// Mitsubishi GX Works2 project: plc_group_3   PLC: FX3G
// 20.11 דורין

// global labels: Global1
VAR_GLOBAL
  START_DAY AT Y010 : BOOL;
  START_WASHING AT X002 : BOOL;
  TS_200 AT TS200 : BOOL;
  Y_5 AT Y005 : BOOL;
  TC_200 AT TC200 : BOOL;
END_VAR
VAR_GLOBAL CONSTANT
  TIMER_1 : INT := 300;
  ORANGE_VALUE : REAL;
END_VAR
VAR_GLOBAL
  ORANGE AT D1270 : REAL;
  ORANGE_STOCK AT D1110 : REAL;  (* ORANGE STOCK *)
  POMELO AT D1280 : REAL;  (* POMELO *)
  POMELO_STOCK AT D1119 : REAL;  (* POMELO *)
  CLAMENTINE AT D1275 : REAL;  (* CLEMENTINE STOCK *)
  CLAMENTINE_wasing AT D1112 : REAL;  (* CLEMENTINE STOCK *)
  POMELO_washing AT D1122 : REAL;  (* POMELO *)
  ORANGE_washing AT D1155 : REAL;
  check_orange_amount AT X020 : BOOL;
  washig_empty AT D1230 : REAL;  (* POMELO *)
  if_more_than_100 AT D1165 : INT;
END_VAR
VAR_GLOBAL CONSTANT
  ORANGES_100 : INT := 100;
END_VAR
VAR_GLOBAL
  OUTPUT_oranges AT D1130 : INT;
  cc_0 AT CC0 : BOOL;
END_VAR
VAR_GLOBAL CONSTANT
  k_2 : WORD := 2;
END_VAR
VAR_GLOBAL
  m_0 AT M0 : BOOL;
  Save_orangeDivideBy2 AT X021 : BOOL;
  ORANGE_amountDivideBy2 AT D1165 : INT;
  ORANGES_DIVIDEby2 AT D1103 : REAL;
END_VAR
VAR_GLOBAL CONSTANT
  DIVIDEby2 : INT := 2;
END_VAR
VAR_GLOBAL
  outC AT CS21 : BOOL;
  firstC AT CC21 : BOOL;
END_VAR
VAR_GLOBAL CONSTANT
  counterK : INT := 3;
END_VAR
VAR_GLOBAL
  coil1 AT Y000 : BOOL;
  cs_0 AT CS0 : BOOL;
  sqeeizing_empty AT D1175 : REAL;  (* POMELO *)
  sqeeizing_start AT D1175 : REAL;  (* sqeeizing *)
  squeezing_juice AT D1130 : REAL;  (* sqeeizing *)
  from_squeezing AT D1135 : REAL;  (* finish_squeezing *)
  new_juice AT D1135 : REAL;  (* juice *)
  move_squeeziToJuice AT D1130 : REAL;  (* juice *)
  get_juice AT D1135 : REAL;  (* juice *)
  X_11 AT X011 : BOOL;
  sub_from_squeezing AT D1130 : REAL;  (* מאפס את מיכל הסחיטה *)
  squeeizing_start AT D1240 : REAL;
  end_squeezing AT M8 : BOOL;
  x_1 AT X001 : BOOL;
  move_oranges_to_squeezing AT D1115 : REAL;  (* sqeeizing *)
END_VAR
VAR_GLOBAL CONSTANT
  empty_juice : REAL;
END_VAR
VAR_GLOBAL
  save_orange_to_squeeze AT D1130 : REAL;
  move_clamentines_to_squeezing AT D1120 : REAL;  (* sqeeizing *)
  move_pomeloes_to_squeezing AT D1125 : REAL;  (* sqeeizing *)
  save_clamentines_to_squeezing AT D1130 : REAL;  (* sqeeizing *)
  save_pomeloes_to_squeezing AT D1130 : REAL;  (* sqeeizing *)
  end_and_start_squeezing AT M7 : BOOL;  (* sqeeizing *)
  finish_help AT M7 : BOOL;
  start_over AT X063 : BOOL;
  Y_1 AT Y001 : BOOL;
  finish_indicator AT Y001 : BOOL;
  CLEMANTINE : REAL;  (* POMELO *)
  CLEMANTINE_STOCK AT D1105 : REAL;
  HELP_ORANGES AT D1165 : REAL;
  HELP_CLEMANTINE AT D1170 : REAL;
  HELP_POMELO AT D1175 : REAL;
  TURN_OFF_X002 AT X002 : BOOL;
  check_quantities_before_transfer AT M8 : BOOL;
  first_mul AT D1190 : REAL;  (* finish_squeezing *)
  RESULT_MUL AT D1195 : REAL;
END_VAR
VAR_GLOBAL CONSTANT
  ZERO : REAL;
  TWO : REAL := 2;
  fifty : REAL := 50;
END_VAR
VAR_GLOBAL
  DOUBLE_POMELO AT D1105 : REAL;
  RESULT_CLEMANTINE AT D1200 : REAL;
  RESULT_POMELO AT D1205 : REAL;
  RESULT_ORANGES AT D1205 : REAL;
END_VAR
VAR_GLOBAL CONSTANT
  HUNDRED : REAL := 100;
END_VAR
VAR_GLOBAL
  DOUBLE_CLEMANTINE AT D1110 : REAL;
  STARTING_switch AT X010 : BOOL;
  CHECK_IF_CORRECT_INPUT AT Y010 : BOOL;
  main_LIGHT AT Y010 : BOOL;
  washig_empty_oranges AT D1230 : REAL;  (* POMELO *)
  washig_empty_pomelo AT D1240 : REAL;  (* POMELO *)
  TC201 : BOOL;
  TC202 : BOOL;
  TC203 : BOOL;
  TC204 : BOOL;
  TC206 : BOOL;
END_VAR
VAR_GLOBAL CONSTANT
  TC207 : INT := 300;
  TC208 : INT := 300;
  TC209 : INT := 300;
END_VAR
VAR_GLOBAL
  TC210 : BOOL;
END_VAR
VAR_GLOBAL CONSTANT
  TC211 : INT := 300;
  TC212 : INT := 300;
  TC213 : INT := 300;
END_VAR
VAR_GLOBAL
  washing_empty_clamentine1 AT D1235 : REAL;  (* POMELO *)
  BLALA AT M5 : BOOL;
  BLA AT M6 : BOOL;
  BLAAA AT M7 : BOOL;
  HELP AT Y100 : BOOL;
  x_1_pulse AT X002 : BOOL;
  quality_check AT X003 : BOOL;
  analog_input_2 AT D8281 : INT;
END_VAR
VAR_GLOBAL CONSTANT
  ONE : REAL := 1;
  five : REAL := 5;
END_VAR
VAR_GLOBAL
  TS_240 AT TS200 : BOOL;
  Y_4 AT Y004 : BOOL;
END_VAR
VAR_GLOBAL CONSTANT
  TIMER_3 : INT := 500;
END_VAR
VAR_GLOBAL
  storage_empty AT D1305 : REAL;
  squeeizing_empty AT D1240 : REAL;
  juice_empty AT D1300 : REAL;
  storage AT D1310 : REAL;
  TC_1 AT TC1 : BOOL;  (* POMELO *)
  TC_2 AT TC2 : BOOL;
END_VAR
VAR_GLOBAL CONSTANT
  sec30 : INT := 30;
END_VAR
VAR_GLOBAL
  TC_27 AT TC27 : BOOL;
  TS_27 AT TS27 : BOOL;
END_VAR
VAR_GLOBAL CONSTANT
  one_sec : INT := 5;
END_VAR
VAR_GLOBAL
  quality_seconed_check AT X003 : BOOL;
  CHECK_IF_ZERO AT M4 : BOOL;
  IS_CORRECT_INPUT : BOOL;
  IF_CORRECT_INPUT AT Y010 : BOOL;
  IF_ORANGES_MORE_THAN_ONE AT M5 : BOOL;
  CHECK_IF_NOT_ZERO AT M4 : BOOL;
  IF_NOT_ZERO AT M4 : BOOL;
  Y_10 AT Y010 : BOOL;
  IF_ZERO AT M4 : BOOL;
  finish_step_one AT M5 : BOOL;
  START_WASH AT X002 : BOOL;
  TC_240 AT TC200 : BOOL;
  Input AT X010 : BOOL;
  CLAMENTINE_STOCK AT D1115 : REAL;  (* CLEMENTINE STOCK *)
  STARTING_DAY AT Y010 : BOOL;
  HELPI AT M8 : BOOL;
  Hghfhfg AT M12 : BOOL;
  HELPU AT Y100 : BOOL;
  m_20 AT M20 : BOOL;
  m_7 AT M21 : BOOL;
  m_25 AT M20 : BOOL;
  m_21 AT M21 : BOOL;
  m_9 AT M0 : BOOL;
  m_15 AT M15 : BOOL;
  sum_washing AT D1450 : REAL;
  m_10 AT M10 : BOOL;
  m_30 AT M30 : BOOL;
  m_31 AT M31 : BOOL;
  m_32 AT M32 : BOOL;
  m_33 AT M33 : BOOL;
  m_34 AT M34 : BOOL;
  m_35 AT M35 : BOOL;
  n_36 AT M36 : BOOL;
  m_36 AT M36 : BOOL;
  m_37 AT M37 : BOOL;
  min_quantity AT D1379 : REAL;
  orange_in_wash AT M32 : BOOL;
  clamentine_in_wash AT M33 : BOOL;  (* CLEMENTINE STOCK *)
  pomelo_in_wash AT M34 : BOOL;  (* POMELO *)
  IF_ZERO_OR_NOT_ENOUGH AT M4 : BOOL;
  m_67 AT M67 : BOOL;
  ORANGE_QUANTITY AT D1865 : REAL;
  QUANTITY_ORANGES AT D1865 : REAL;
  Y_7 AT Y007 : BOOL;
END_VAR
VAR_GLOBAL CONSTANT
  TRUE1 : BOOL := TRUE;
END_VAR
VAR_GLOBAL
  x_3 AT X003 : BOOL;
END_VAR
VAR_GLOBAL CONSTANT
  DIV_400 : REAL := 400;
END_VAR
VAR_GLOBAL
  analog_val AT D4000 : REAL;
  m_40 AT M40 : BOOL;
  m_43 AT M43 : BOOL;
  T_4 AT M445 : BOOL;
END_VAR
VAR_GLOBAL CONSTANT
  const_5 : REAL := 5;
END_VAR
VAR_GLOBAL
  m_41 AT M41 : BOOL;
END_VAR
VAR_GLOBAL CONSTANT
  constant_1 : REAL := 1;
END_VAR
VAR_GLOBAL
  m_42 AT M42 : BOOL;
END_VAR
VAR_GLOBAL CONSTANT
  seconds_5 : INT := 500;
END_VAR
VAR_GLOBAL
  TC_4 AT TC4 : BOOL;  (* POMELO *)
  TS_4 AT TS4 : BOOL;
  TC_205 AT TC205 : BOOL;
  TS_205 AT TS205 : BOOL;
END_VAR
VAR_GLOBAL CONSTANT
  const_2 : INT := 2;
END_VAR
VAR_GLOBAL
  TC_206 AT TC206 : BOOL;
  TS_206 AT TS206 : BOOL;
  cc_1 AT CC1 : BOOL;
  cs_1 AT CS1 : BOOL;
  m_44 AT M44 : BOOL;
  GT_result : BOOL;
  m_45 AT M45 : BOOL;
END_VAR
VAR_GLOBAL CONSTANT
  const_1 : INT := 1;
  Bit_on : BOOL := TRUE;
END_VAR
VAR_GLOBAL
  m_46 AT M46 : BOOL;
  analog_output AT D8282 : INT;
  x_6 AT X006 : BOOL;
  TC_201 AT TC201 : BOOL;
  TS_201 AT TS201 : BOOL;
END_VAR
VAR_GLOBAL CONSTANT
  const_0 : INT;
  const_15 : INT := 10;
END_VAR
VAR_GLOBAL
  temperature AT D5001 : INT;
END_VAR
VAR_GLOBAL CONSTANT
  mol_400 : INT := 400;
END_VAR
VAR_GLOBAL
  m_11 AT M11 : BOOL;
END_VAR
VAR_GLOBAL CONSTANT
  const_10 : INT := 10;
END_VAR
VAR_GLOBAL
  CLAMENTINE_washing AT D1112 : REAL;  (* CLEMENTINE STOCK *)
  x_7 AT X007 : BOOL;
  emergancy_switch AT M7 : BOOL;  (* sqeeizing *)
  m_13 AT M13 : BOOL;
  m_50 AT M50 : BOOL;
  m_51 AT M51 : BOOL;
  Y_2 AT Y002 : BOOL;
  Y_3 AT Y003 : BOOL;
  m_22 AT M22 : BOOL;
  m_55 AT M55 : BOOL;
END_VAR
VAR_GLOBAL CONSTANT
  TIMER_washing : INT := 300;
END_VAR
VAR_GLOBAL
  m_60 AT M60 : BOOL;
  M_61 AT M61 : BOOL;
  sum_storage AT D7146 : REAL;
  M_63 AT M63 : BOOL;
  m_12 AT M12 : BOOL;
  m_52 AT M52 : BOOL;
  M_4 : BOOL;
  m_79 AT M79 : BOOL;
END_VAR
VAR_GLOBAL CONSTANT
  TIMER_2 : INT := 300;
END_VAR
VAR_GLOBAL
  TC_204 AT TC204 : BOOL;
  m_19 AT M19 : BOOL;
  TC_6 AT TC6 : BOOL;
END_VAR
VAR_GLOBAL CONSTANT
  false1 : BOOL;
END_VAR
VAR_GLOBAL
  m_47 AT M47 : BOOL;
END_VAR

// task Task_01 (event TRUE, interval 0, priority 31): POU_01

PROGRAM POU_01
(* structured ladder/FBD written out as ST: instructions are called as NAME(EN, inputs, outputs); _pN, _eN, _tN stand for wires *)
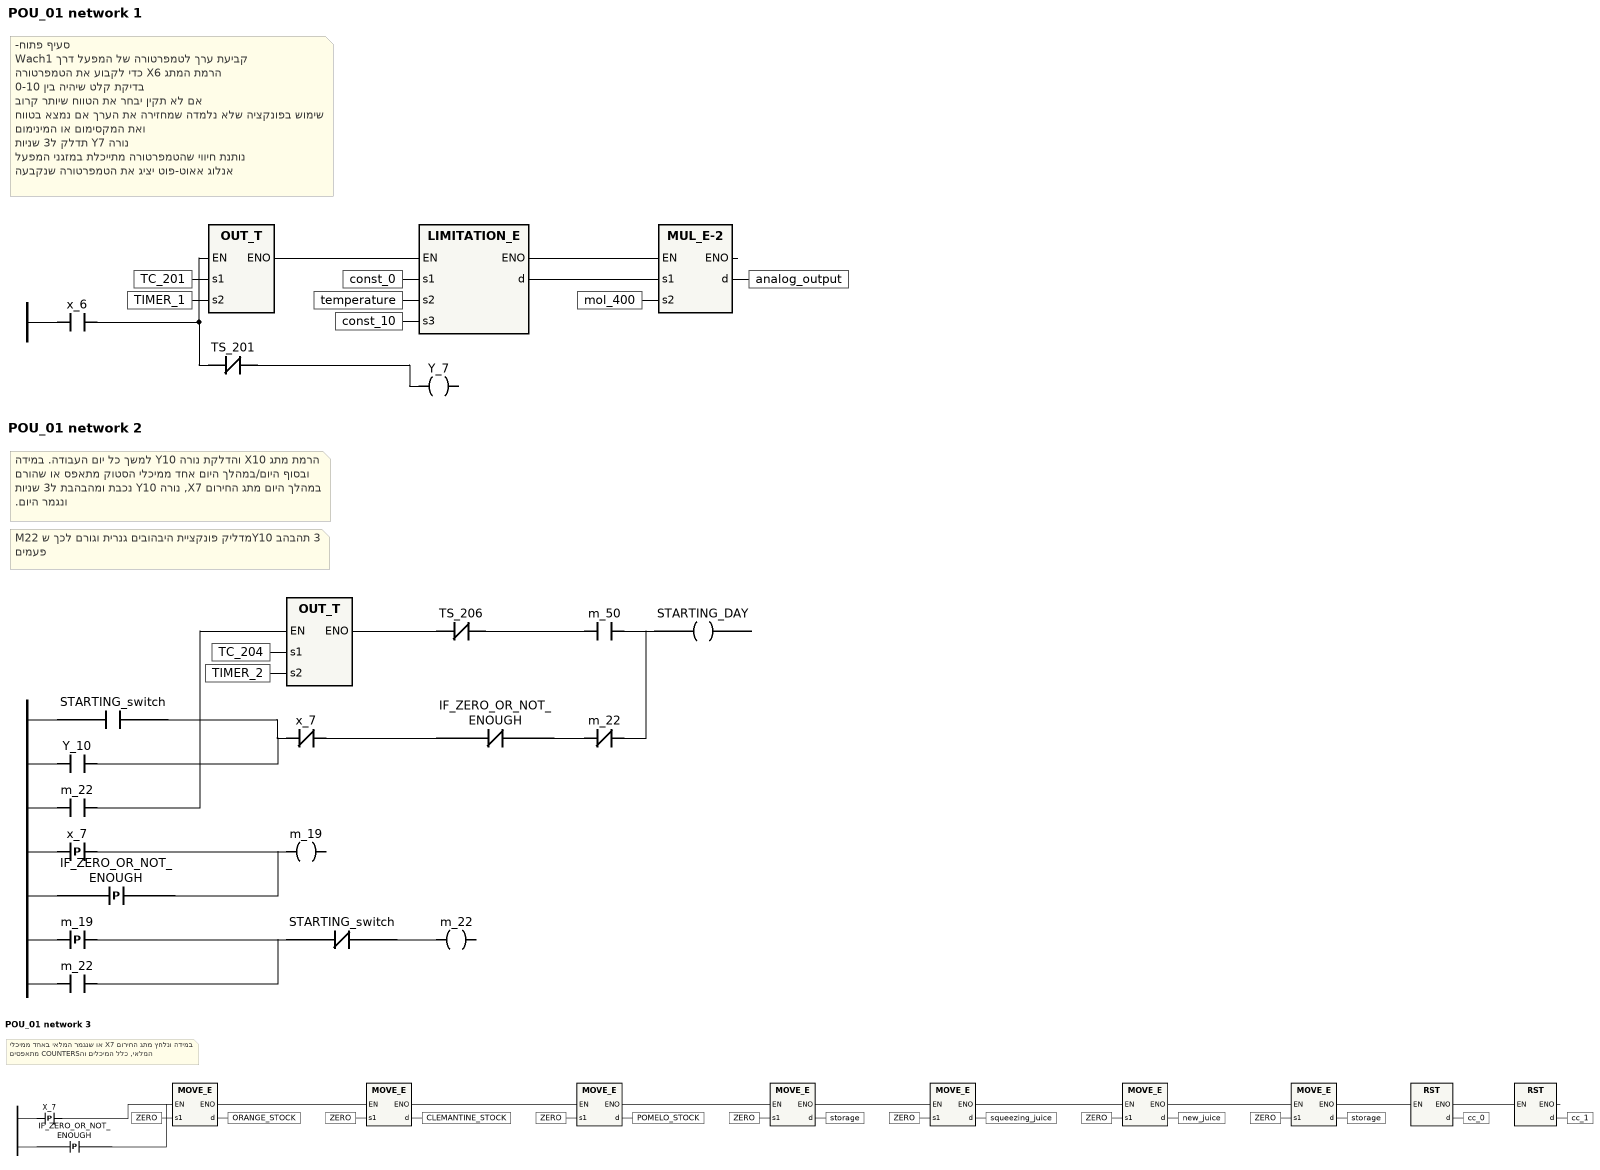
(* network 1 *)
(* סעיף פתוח- / קביעת ערך לטמפרטורה של המפעל דרך Wach1  / הרמת המתג X6 כדי לקבוע את הטמפרטורה / בדיקת קלט שיהיה בין 0-10  / אם לא תקין יבחר את הטווח שיותר קרוב  / שימוש בפונקציה שלא נלמדה שמחזירה את הערך אם נמצא בטווח ואת המקסימום או המינימום  / נורה Y7 תדלק ל3 שניות  / נותנת חיווי שהטמפרטורה מתייכלת במזגני המפעל  / אנלוג אאוט-פוט יציג את הטמפרטורה שנקבעה *)
_e1 := OUT_T(x_6, TC_201, TIMER_1);
_e3 := LIMITATION_E(_e1, const_0, temperature, const_10, _t2);
MUL_E(_e3, _t2, mol_400, analog_output);
Y_7 := x_6 AND NOT TS_201;
(* network 2 *)
(* הרמת מתג X10 והדלקת נורה Y10 למשך כל יום העבודה. במידה ובסוף היום/במהלך היום אחד ממיכלי הסטוק מתאפס או שהורם במהלך היום מתג החירום X7, נורה Y10 נכבת ומהבהבת ל3 שניות ונגמר היום. *)
(* M22 מדליק פונקציית היבהובים גנרית וגורם לכך שY10 תהבהב 3 פעמים *)
_e1 := OUT_T(m_22, TC_204, TIMER_2);
STARTING_DAY := ((((STARTING_switch OR Y_10) AND NOT x_7) AND NOT IF_ZERO_OR_NOT_ENOUGH) AND NOT m_22) OR (_e1 AND NOT TS_206 AND m_50);
m_19 := LDP(TRUE, x_7) OR LDP(TRUE, IF_ZERO_OR_NOT_ENOUGH);
m_22 := (LDP(TRUE, m_19) OR m_22) AND NOT STARTING_switch;
(* network 3 *)
(* במידה ונלחץ מתג החירום X7 או שנגמר המלאי באחד ממיכלי המלאי, כלל המיכלים והCOUNTERS מתאפסים *)
_e1 := MOVE_E(LDP(TRUE, X_7) OR LDP(TRUE, IF_ZERO_OR_NOT_ENOUGH), ZERO, ORANGE_STOCK);
_e2 := MOVE_E(_e1, ZERO, CLEMANTINE_STOCK);
_e3 := MOVE_E(_e2, ZERO, POMELO_STOCK);
_e4 := MOVE_E(_e3, ZERO, storage);
_e5 := MOVE_E(_e4, ZERO, squeezing_juice);
_e6 := MOVE_E(_e5, ZERO, new_juice);
_e7 := MOVE_E(_e6, ZERO, storage);
_e8 := RST(_e7, cc_0);
RST(_e8, cc_1);
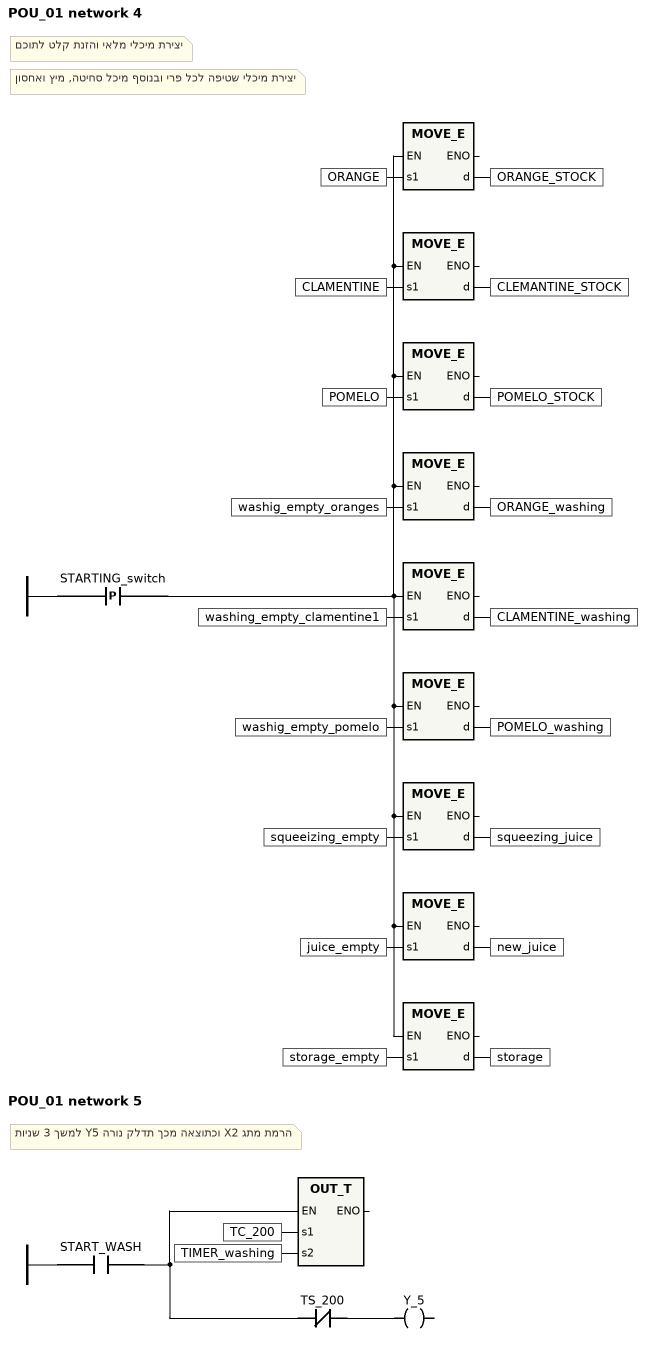
(* network 4 *)
(* יצירת מיכלי מלאי והזנת קלט לתוכם *)
(* יצירת מיכלי שטיפה לכל פרי ובנוסף מיכל סחיטה, מיץ ואחסון *)
_p1 := LDP(TRUE, STARTING_switch);
MOVE_E(_p1, ORANGE, ORANGE_STOCK);
MOVE_E(_p1, CLAMENTINE, CLEMANTINE_STOCK);
MOVE_E(_p1, POMELO, POMELO_STOCK);
MOVE_E(_p1, washig_empty_oranges, ORANGE_washing);
MOVE_E(_p1, washing_empty_clamentine1, CLAMENTINE_washing);
MOVE_E(_p1, washig_empty_pomelo, POMELO_washing);
MOVE_E(_p1, squeeizing_empty, squeezing_juice);
MOVE_E(_p1, juice_empty, new_juice);
MOVE_E(_p1, storage_empty, storage);
(* network 5 *)
(* הרמת מתג X2 וכתוצאה מכך תדלק נורה Y5 למשך 3 שניות *)
OUT_T(START_WASH, TC_200, TIMER_washing);
Y_5 := START_WASH AND NOT TS_200;
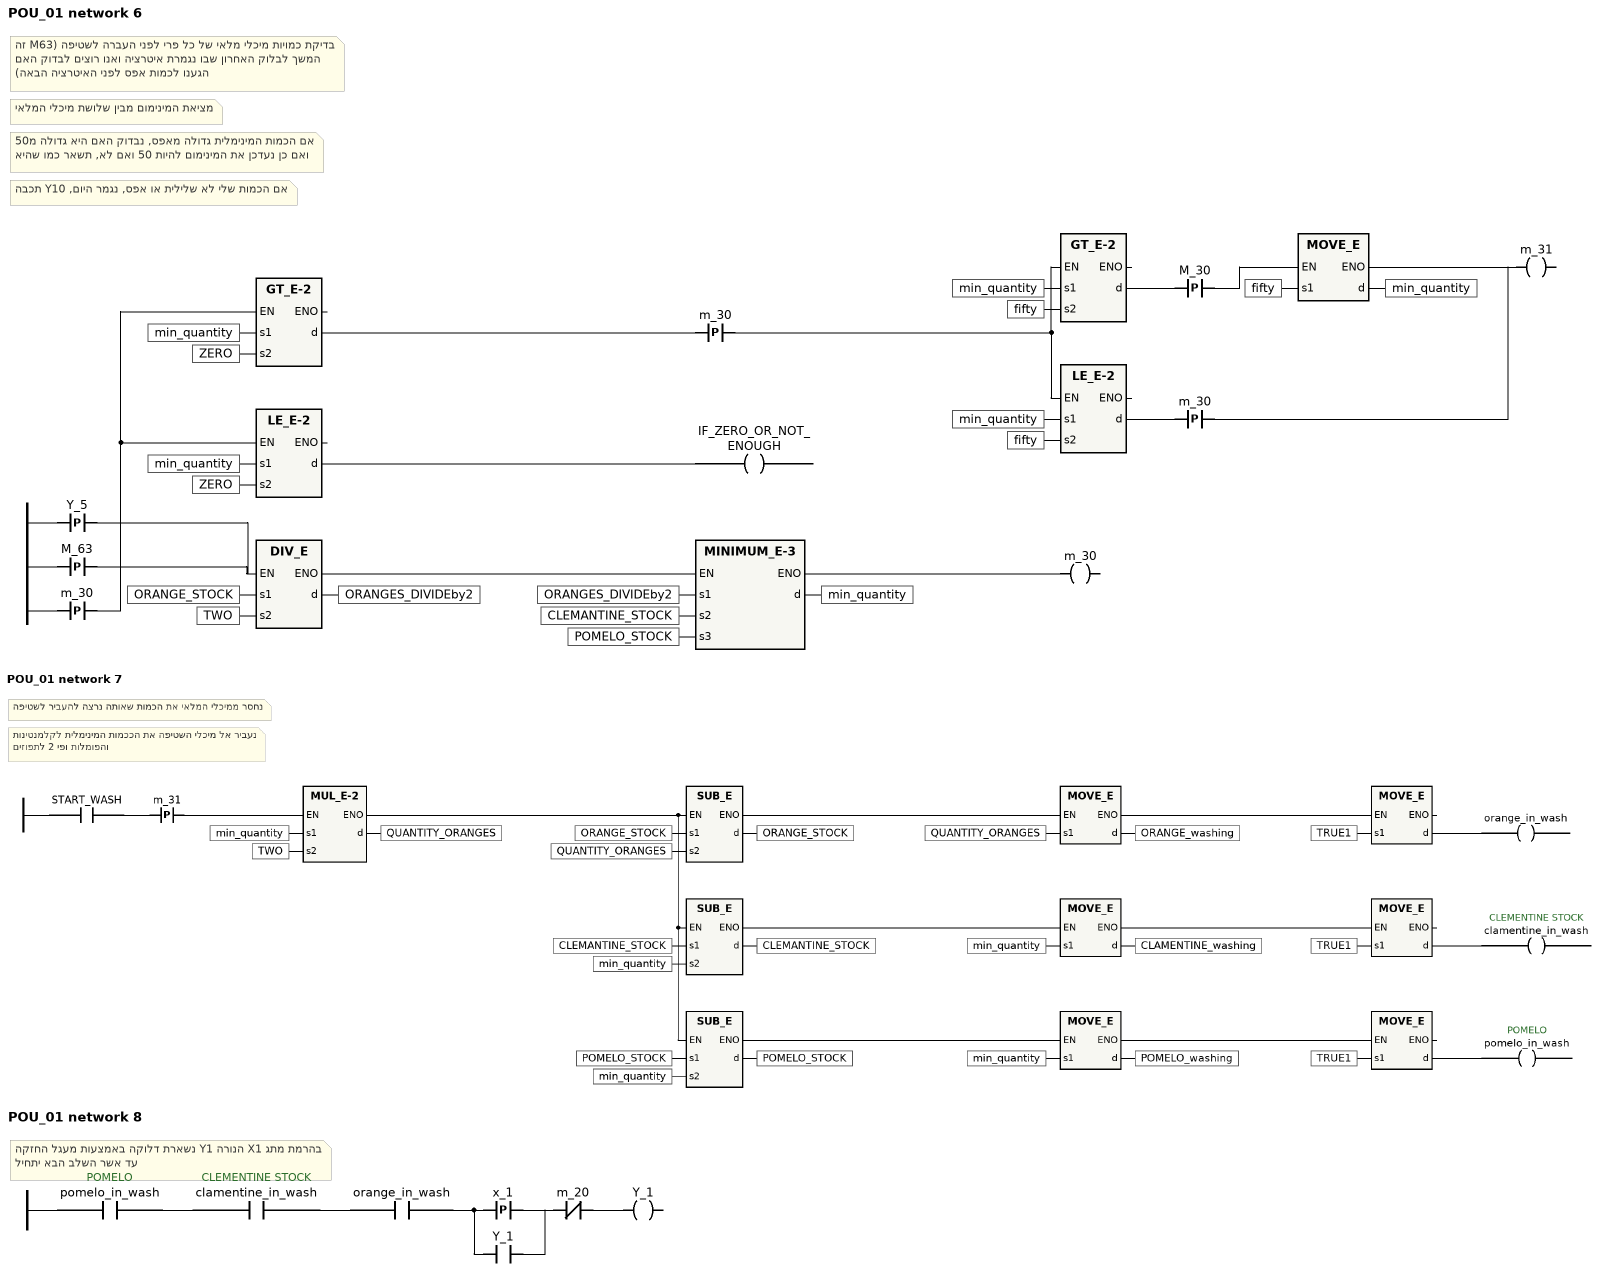
(* network 6 *)
(* בדיקת כמויות מיכלי מלאי של כל פרי לפני העברה לשטיפה (M63 זה המשך לבלוק האחרון שבו נגמרת איטרציה ואנו רוצים לבדוק האם הגענו לכמות אפס לפני האיטרציה הבאה) *)
(* מציאת המינימום מבין שלושת מיכלי המלאי *)
(* אם הכמות המינימלית גדולה מאפס, נבדוק האם היא גדולה מ50 ואם כן נעדכן את המינימום להיות 50 ואם לא, תשאר כמו שהיא *)
(* אם הכמות שלי לא שלילית או אפס, נגמר היום, Y10 תכבה *)
_e1 := DIV_E(LDP(TRUE, Y_5) OR LDP(TRUE, M_63), ORANGE_STOCK, TWO, ORANGES_DIVIDEby2);
_e2 := MINIMUM_E(_e1, ORANGES_DIVIDEby2, CLEMANTINE_STOCK, POMELO_STOCK, min_quantity);
m_30 := _e2;
_p3 := LDP(TRUE, m_30);
GT_E(_p3, min_quantity, ZERO, _t4);
_p5 := _t4 AND LDP(TRUE, m_30);
GT_E(_p5, min_quantity, fifty, _t6);
_e7 := MOVE_E(_t6 AND LDP(TRUE, M_30), fifty, min_quantity);
LE_E(_p5, min_quantity, fifty, _t8);
m_31 := _e7 OR (_t8 AND LDP(TRUE, m_30));
LE_E(_p3, min_quantity, ZERO, _t9);
IF_ZERO_OR_NOT_ENOUGH := _t9;
(* network 7 *)
(* נחסר ממיכלי המלאי את הכמות שאותה נרצה להעביר לשטיפה *)
(* נעביר אל מיכלי השטיפה את הככמות המינימלית לקלמנטינות והפומלות ופי 2 לתפוזים *)
_e1 := MUL_E(START_WASH AND LDP(TRUE, m_31), min_quantity, TWO, QUANTITY_ORANGES);
_e2 := SUB_E(_e1, ORANGE_STOCK, QUANTITY_ORANGES, ORANGE_STOCK);
_e3 := MOVE_E(_e2, QUANTITY_ORANGES, ORANGE_washing);
MOVE_E(_e3, TRUE1, _t4);
orange_in_wash := _t4;
_e5 := SUB_E(_e1, CLEMANTINE_STOCK, min_quantity, CLEMANTINE_STOCK);
_e6 := MOVE_E(_e5, min_quantity, CLAMENTINE_washing);
MOVE_E(_e6, TRUE1, _t7);
clamentine_in_wash := _t7;
_e8 := SUB_E(_e1, POMELO_STOCK, min_quantity, POMELO_STOCK);
_e9 := MOVE_E(_e8, min_quantity, POMELO_washing);
MOVE_E(_e9, TRUE1, _t10);
pomelo_in_wash := _t10;
(* network 8 *)
(* בהרמת מתג X1 הנורה Y1 נשארת דלוקה באמצעות מעגל החזקה עד אשר השלב הבא יתחיל *)
_p1 := pomelo_in_wash AND clamentine_in_wash AND orange_in_wash;
Y_1 := ((_p1 AND LDP(TRUE, x_1)) OR (_p1 AND Y_1)) AND NOT m_20;
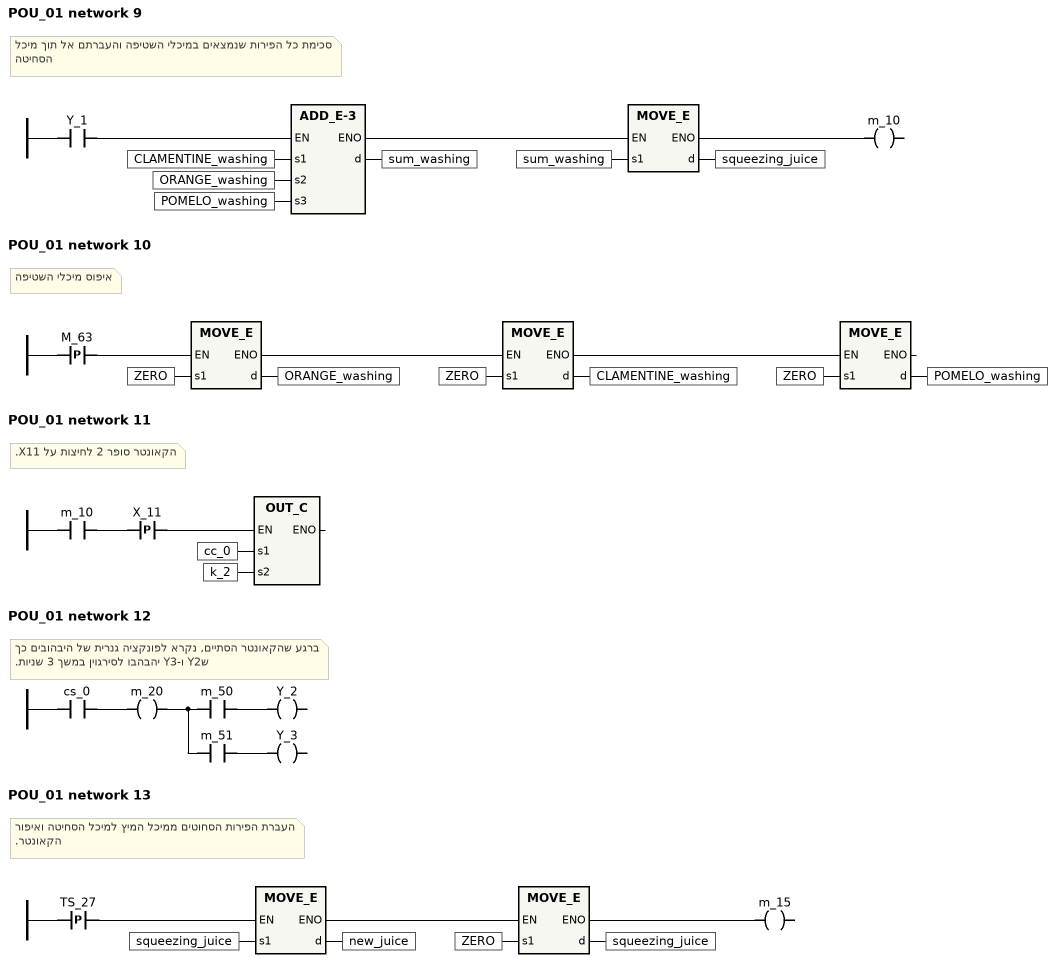
(* network 9 *)
(* סכימת כל הפירות שנמצאים במיכלי השטיפה והעברתם אל תוך מיכל הסחיטה *)
_e1 := ADD_E(Y_1, CLAMENTINE_washing, ORANGE_washing, POMELO_washing, sum_washing);
_e2 := MOVE_E(_e1, sum_washing, squeezing_juice);
m_10 := _e2;
(* network 10 *)
(* איפוס מיכלי השטיפה *)
_e1 := MOVE_E(LDP(TRUE, M_63), ZERO, ORANGE_washing);
_e2 := MOVE_E(_e1, ZERO, CLAMENTINE_washing);
MOVE_E(_e2, ZERO, POMELO_washing);
(* network 11 *)
(* הקאונטר סופר 2 לחיצות על X11. *)
OUT_C(m_10 AND LDP(TRUE, X_11), cc_0, k_2);
(* network 12 *)
(* ברגע שהקאונטר הסתיים, נקרא לפונקציה גנרית של היבהובים כך שY2 ו-Y3 יהבהבו לסירגוין במשך 3 שניות. *)
m_20 := cs_0;
Y_2 := cs_0 AND m_50;
Y_3 := cs_0 AND m_51;
(* network 13 *)
(* העברת הפירות הסחוטים ממיכל המיץ למיכל הסחיטה ואיפור הקאונטר. *)
_e1 := MOVE_E(LDP(TRUE, TS_27), squeezing_juice, new_juice);
_e2 := MOVE_E(_e1, ZERO, squeezing_juice);
m_15 := _e2;
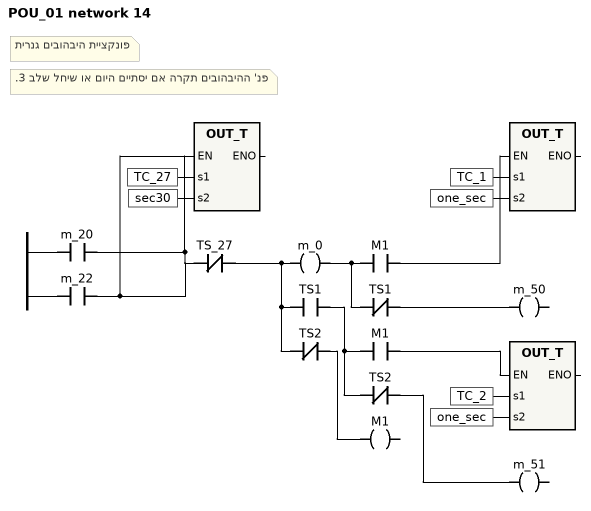
(* network 14 *)
(* פונקציית היבהובים גנרית *)
(* פנ' ההיבהובים תקרה אם יסתיים היום או שיחל שלב 3. *)
_p1 := m_20 OR m_22;
OUT_T(_p1, TC_27, sec30);
_p2 := _p1 AND NOT TS_27;
m_0 := _p2;
OUT_T(_p2 AND M1, TC_1, one_sec);
m_50 := _p2 AND NOT TS1;
_p3 := _p2 AND TS1;
OUT_T(_p3 AND M1, TC_2, one_sec);
m_51 := _p3 AND NOT TS2;
M1 := _p2 AND NOT TS2;
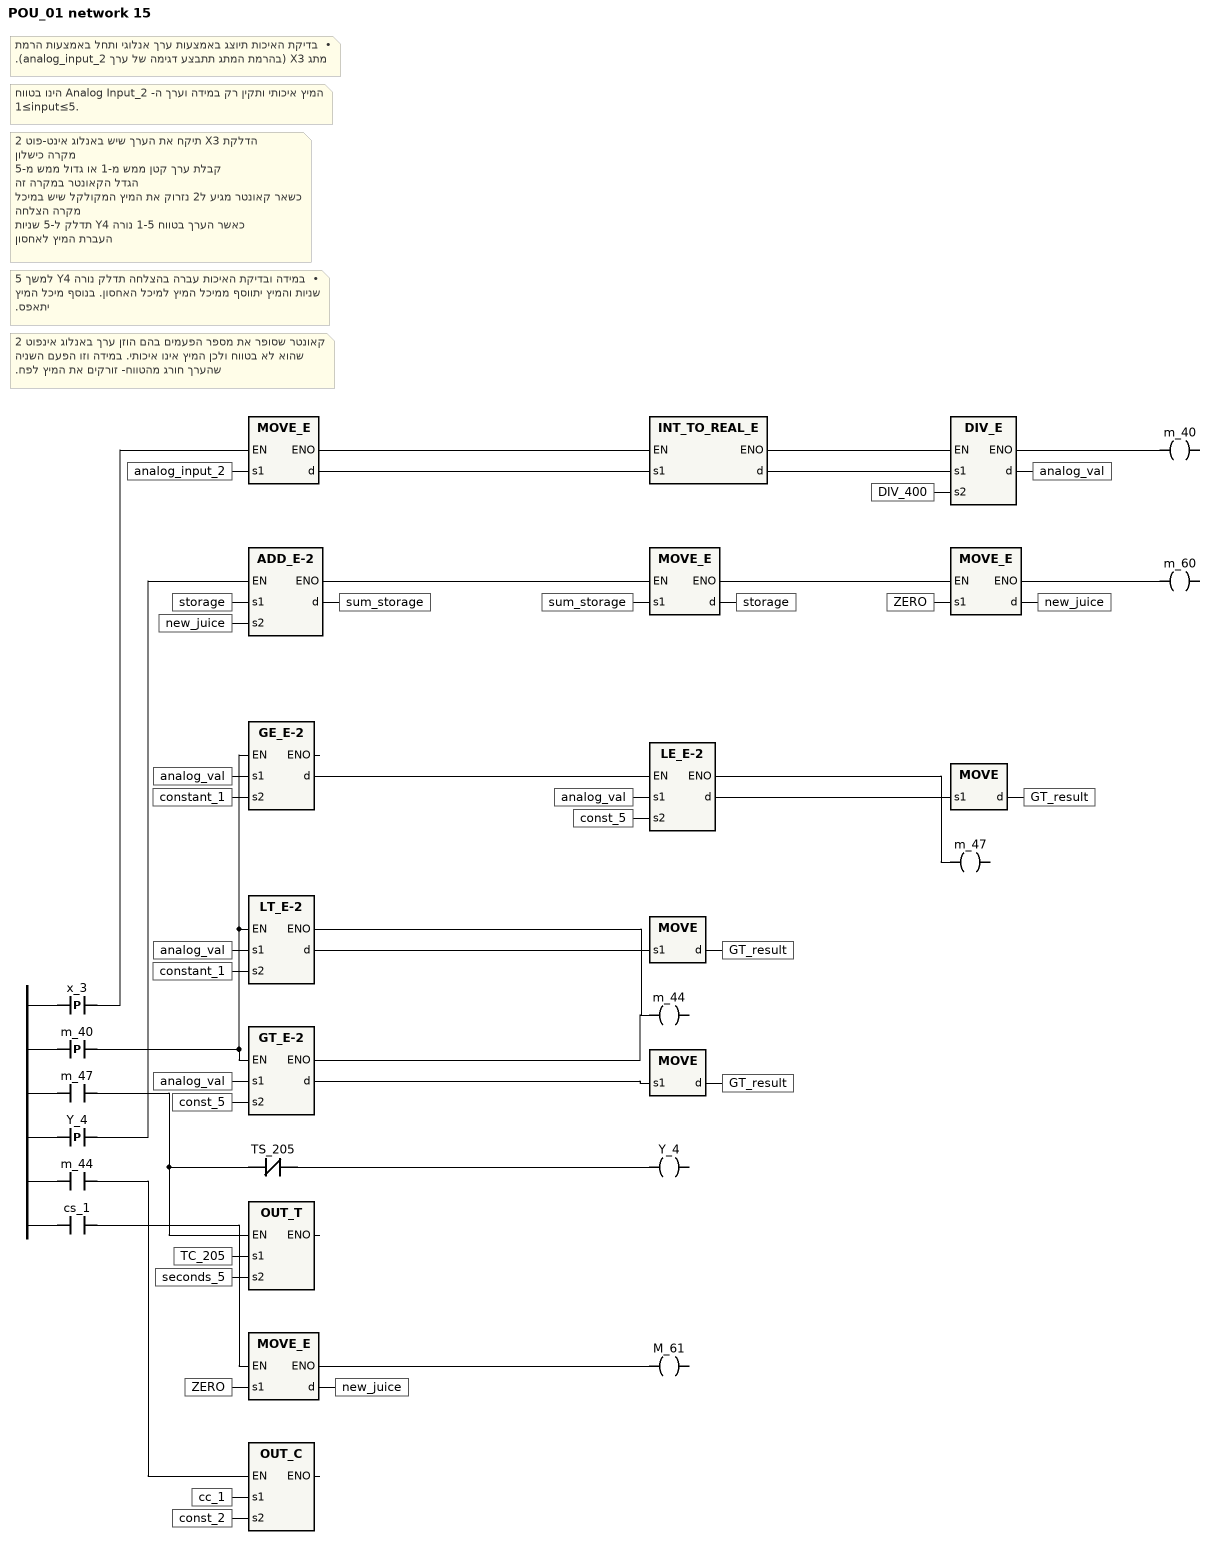
(* network 15 *)
(* •	בדיקת האיכות תיוצג באמצעות ערך אנלוגי ותחל באמצעות הרמת מתג X3 (בהרמת המתג תתבצע דגימה של ערך analog_input_2). *)
(* המיץ איכותי ותקין רק במידה וערך ה- Analog Input_2 הינו בטווח 1≤input≤5. *)
(* הדלקת X3 תיקח את הערך שיש באנלוג אינט-פוט 2 /  / מקרה כישלון /  / קבלת ערך קטן ממש מ-1 או גדול ממש מ-5 / הגדל הקאונטר במקרה זה / כשאר קאונטר מגיע ל2 נזרוק את המיץ המקולקל שיש במיכל /  /  / מקרה הצלחה / כאשר הערך בטווח 1-5 נורה Y4 תדלק ל-5 שניות / העברת המיץ לאחסון *)
(* •	במידה ובדיקת האיכות עברה בהצלחה תדלק נורה Y4 למשך 5 שניות והמיץ יתווסף ממיכל המיץ למיכל האחסון. בנוסף מיכל המיץ יתאפס. *)
(* קאונטר שסופר את מספר הפעמים בהם הוזן ערך באנלוג אינפוט 2 שהוא לא בטווח ולכן המיץ אינו איכותי. במידה וזו הפעם השניה שהערך חורג מהטווח- זורקים את המיץ לפח. *)
_e2 := MOVE_E(LDP(TRUE, x_3), analog_input_2, _t1);
_e4 := INT_TO_REAL_E(_e2, _t1, _t3);
_e5 := DIV_E(_e4, _t3, DIV_400, analog_val);
m_40 := _e5;
_p6 := LDP(TRUE, m_40);
GE_E(_p6, analog_val, constant_1, _t7);
_e9 := LE_E(_t7, analog_val, const_5, _t8);
m_47 := _e9;
GT_result := MOVE(_t8);
_e11 := LT_E(_p6, analog_val, constant_1, _t10);
GT_result := MOVE(_t10);
_e13 := GT_E(_p6, analog_val, const_5, _t12);
m_44 := _e11 OR _e13;
GT_result := MOVE(_t12);
OUT_T(m_47, TC_205, seconds_5);
Y_4 := m_47 AND NOT TS_205;
_e14 := ADD_E(LDP(TRUE, Y_4), storage, new_juice, sum_storage);
_e15 := MOVE_E(_e14, sum_storage, storage);
_e16 := MOVE_E(_e15, ZERO, new_juice);
m_60 := _e16;
OUT_C(m_44, cc_1, const_2);
_e17 := MOVE_E(cs_1, ZERO, new_juice);
M_61 := _e17;
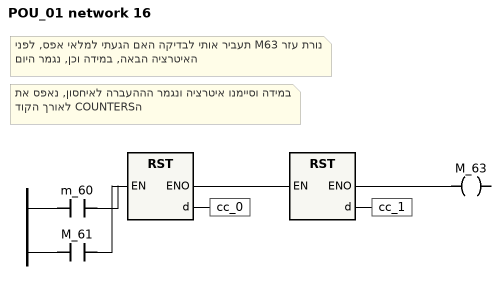
(* network 16 *)
(* נורת עזר M63 תעביר אותי לבדיקה האם הגעתי למלאי אפס, לפני האיטרציה הבאה, במידה וכן, נגמר היום *)
(* במידה וסיימנו איטרציה ונגמר הההעברה לאיחסון, נאפס את הCOUNTERS לאורך הקוד *)
_e1 := RST(m_60 OR M_61, cc_0);
_e2 := RST(_e1, cc_1);
M_63 := _e2;
END_PROGRAM
